// Processor used by the machine.
{attribute 'qualified_only'}
{attribute 'to_string'}
TYPE E_ProcessorArchitecture :
(
	_ 			:= 0, 	// Invalid/Unknown/Ininitialised
	X86,				// X86 Processor
	ARM,				// ARM Processor
	PowerPC,			// PowerPC Processor
	MIPS				// MIPS processor (as of March 2021 MIPS Technology has moved to RISC-V)
)BYTE;
END_TYPE

(* stored: Version 1.1.0.1
   EnumerationTextList E_ProcessorArchitecture: Id {babaeb39-6251-0881-2c61-3df69b27dcc3} *)
